// TIA Portal V16 export
// export: Created 2020-03-07T17:54:54.5356049Z, ExportSetting WithDefaults, DisplayName Totally Integrated Automation Portal, DisplayVersion V16 Update 1, DisplayName TIA Portal Version Control Interface, DisplayVersion V16, DisplayName TIA Portal Openness, DisplayVersion V16 Update 1, DisplayName STEP 7 Professional, DisplayVersion V16 Update 1, DisplayName STEP 7 Safety, DisplayVersion V16, DisplayName WinCC Professional, DisplayVersion V16 Update 1
DATA_BLOCK "Data_block_1"   // DB2
{ S7_Optimized_Access := 'TRUE' }
VERSION : 0.1
// stored: AutoNumber true, DBAccessibleFromOPCUA true, IsOnlyStoredInLoadMemory false, IsRetainMemResEnabled false, IsWriteProtectedInAS false, MemoryReserve 0
   VAR
      x : Bool;
      y : Bool;
      z : Bool;
      fc1_edge : Bool;
      fc1_catch_signal : Bool;
      fc1_output : Bool;
      "a" : Int;
      "b" : Int;
      c : Int;
      d : Int;
   END_VAR
BEGIN
END_DATA_BLOCK
